{attribute 'Tc2GvlVarNames'}
VAR_GLOBAL
	IN_Stromzaehler AT %I* 	: ST_KL6781inData22B;
	OUT_Stromzaehler AT %Q* : ST_KL6781outData22B;
	IN_WZaehler AT %I* 	: ST_KL6781inData22B;
	OUT_WZaehler AT %Q* : ST_KL6781outData22B;
	
	//container
	HeatCounters_Container_IN AT %I* : ST_KL6781inData22B;
	HeatCounters_Container_OUT AT %Q* : ST_KL6781outData22B;
	
	(*
			[1] ETA_3111U1006XHE321XXXXXXZ01, ELT_Zaehler_BHKW_321_01
			Primaer-Adresse = 1
			Seriennummer = 3999427
			[2] ETA_3111U1006XHE322XXXXXXZ01, ELT_Zaehler_BHKW_322_01
			Primaer-Adresse = 2
			Seriennummer = 3999432
			[3] ETA_3111U1006BEST001XXXXXXZ01, ELT_Zaehler_Buerotrakt_01
			Primaer-Adresse = 3
			Seriennummer = 120267
			[4] ETA_3111U1006BEST002XXXXXXZ01, ELT_Zaehler_Gebaede_01
			Primaer-Adresse = 4
			Seriennummer = 205684
			[5] ETA_3111U1006BEST003XXXXXXZ01, ELT_Zaehler_Halle_TGA_01
			Primaer-Adresse = 5
			Seriennummer = 120264
			[6] ETA_3111EG005BEST004XXXXXXZ01, ELT_Zaehler_Halle_Licht_01
			Primaer-Adresse = 6
			Seriennummer = 214516
			[7] ETA_3111U1006BEST007XXXXXXZ01, GAS_Zaehler BHKW_007_01
			Primaer-Adresse = 7
			Seriennummer = 42078747
			[8] ETA_3111U1006BEST008XXXXXXZ01, GAS_Zaehler BHKW_008_01
			Primaer-Adresse = 8
			Seriennummer = 42078748
			[9] ETA_3111U1006BEST071XXXXXXZ01, WAERME_Zaehler WP_945_4371_01
			Primaer-Adresse = 71
			Seriennummer = 67694371
			[10] ETA_3111U1006BEST072XXXXXXZ01, WAERME_Zaehler WP_945_4372_01
			Primaer-Adresse = 72
			Seriennummer = 67694372
	*)
	Kommunikation_MBus	: ST_MBUS_Communication;
	Komm_MBus_WZaehler	: ST_MBUS_Communication;

	Telegramm_WZ_Brennwerttherme			: ARRAY[1..cMBUS_MaxTelegrams] OF ST_MBus_Data2;
	Telegramm_WZ_BHKW_1						: ARRAY[1..cMBUS_MaxTelegrams] OF ST_MBus_Data2;
	Telegramm_WZ_BHKW_2						: ARRAY[1..cMBUS_MaxTelegrams] OF ST_MBus_Data2;
	Telegramm_WZ_Druckluftkompressor		: ARRAY[1..cMBUS_MaxTelegrams] OF ST_MBus_Data2;
	Telegramm_WZ_PWT_1						: ARRAY[1..cMBUS_MaxTelegrams] OF ST_MBus_Data2;
	Telegramm_WZ_Ofenkuehlung				: ARRAY[1..cMBUS_MaxTelegrams] OF ST_MBus_Data2;
	Telegramm_WZ_Abwaerme_Ofen_Abgasfackel	: ARRAY[1..cMBUS_MaxTelegrams] OF ST_MBus_Data2;
	
	//heat counters container
	aCommunication_MBus_Container : ST_MBUS_Communication;
	aTelegramm_WMZ138 : ARRAY[1..cMBUS_MaxTelegrams] OF ST_MBus_Data2;

	Telegramm_SZ_BHKW_321		: ARRAY[1..cMBUS_MaxTelegrams] OF ST_MBus_Data2;
	Telegramm_SZ_BHKW_322		: ARRAY[1..cMBUS_MaxTelegrams] OF ST_MBus_Data2;
	Telegramm_SZ_Buerotrakt		: ARRAY[1..cMBUS_MaxTelegrams] OF ST_MBus_Data2;
	Telegramm_SZ_Gebaeude		: ARRAY[1..cMBUS_MaxTelegrams] OF ST_MBus_Data2;
	Telegramm_SZ_Halle_TGA		: ARRAY[1..cMBUS_MaxTelegrams] OF ST_MBus_Data2;
	Telegramm_SZ_Halle_Licht	: ARRAY[1..cMBUS_MaxTelegrams] OF ST_MBus_Data2;

	Telegramm_GZ_BHKW_321		: ARRAY[1..cMBUS_MaxTelegrams] OF ST_MBus_Data2;
	Telegramm_GZ_BHKW_322		: ARRAY[1..cMBUS_MaxTelegrams] OF ST_MBus_Data2;

	Telegramm_WZ_4371_WP_946	: ARRAY[1..cMBUS_MaxTelegrams] OF ST_MBus_Data2;
	Telegramm_WZ_4372_WP_946	: ARRAY[1..cMBUS_MaxTelegrams] OF ST_MBus_Data2;

END_VAR

(* stored: Version 1.1.0.1, ProductVersion 3.1.4024.10
   GVL M_Bus: Id {09f3b77d-e1a8-4a2e-b9d8-80d0df79e368} *)
